TYPE "PositioningMachine_Manager"
VERSION : 0.1
// Block: PositioningMachine_Manager
   STRUCT
      EnableStopDoorOpeningReq : Bool;
      EnableStopInPhase : Bool;
      EnableStopProgrammed : Bool;
      Control_ON : Bool;
      SelectMotorEncoder : Bool;
      Bwd : Bool;
      Fwd : Bool;
      MoveToPos : Bool;
      UsePositionControl : Bool;
      Pos : LReal;
      Vel : LReal;
      Acc : LReal;
      Dec : LReal;
      Jerk : LReal;
   END_STRUCT;

END_TYPE
